// LS Electric XG5000 project: Test1108
// PLC NewPLC
// module base 0 slot 0: 입출력 모듈:XBC-DR32H (DC 24V 입력, 릴레이 출력 32점)

PROGRAM NewProgram (task: 스캔 프로그램)

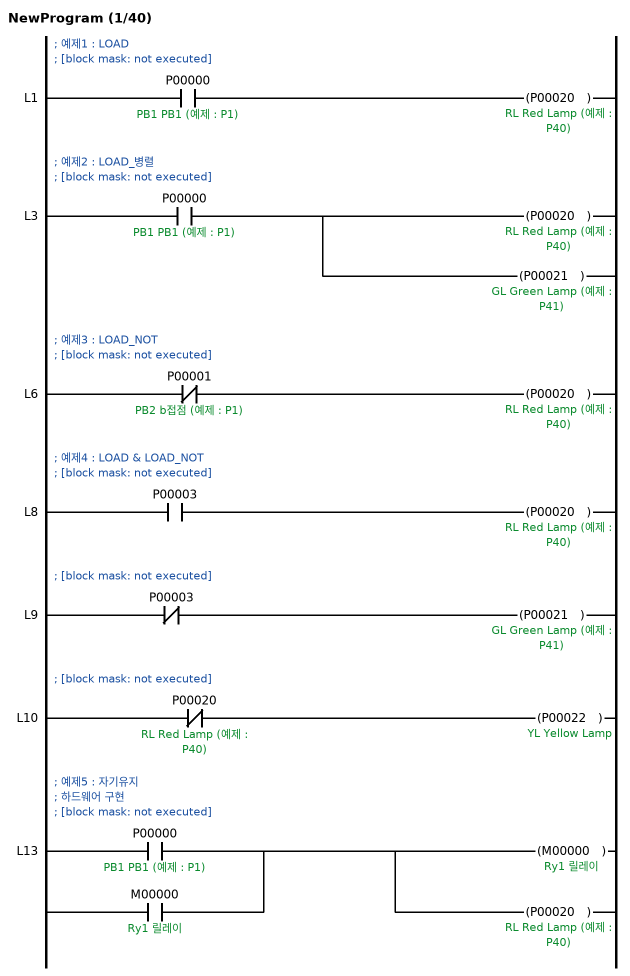
// 예제1 : LOAD
; L1 (block mask: not executed)
LOAD      P00000	// PB1 PB1 (예제 : P1)
OUT       P00020	// RL Red Lamp (예제 : P40)
// 예제2 : LOAD_병렬
; L3 (block mask: not executed)
LOAD      P00000	// PB1 PB1 (예제 : P1)
OUT       P00020	// RL Red Lamp (예제 : P40)
OUT       P00021	// GL Green Lamp (예제 : P41)
// 예제3 : LOAD_NOT 
; L6 (block mask: not executed)
LOAD NOT  P00001	// PB2 b접점 (예제 : P1)
OUT       P00020	// RL Red Lamp (예제 : P40)
// 예제4 : LOAD & LOAD_NOT
; L8 (block mask: not executed)
LOAD      P00003
OUT       P00020	// RL Red Lamp (예제 : P40)
; L9 (block mask: not executed)
LOAD NOT  P00003
OUT       P00021	// GL Green Lamp (예제 : P41)
; L10 (block mask: not executed)
LOAD NOT  P00020	// RL Red Lamp (예제 : P40)
OUT       P00022	// YL Yellow Lamp
// 예제5 : 자기유지
// 하드웨어 구현
; L13 (block mask: not executed)
LOAD      P00000	// PB1 PB1 (예제 : P1)
OR        M00000	// Ry1 릴레이
OUT       M00000	// Ry1 릴레이
OUT       P00020	// RL Red Lamp (예제 : P40)

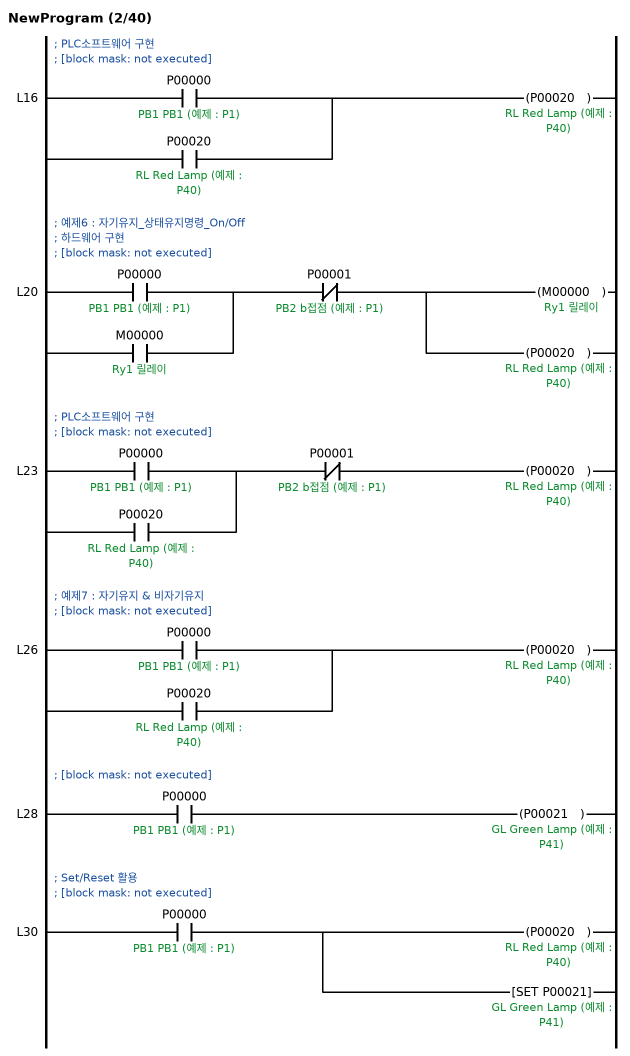
// PLC소프트웨어 구현
; L16 (block mask: not executed)
LOAD      P00000	// PB1 PB1 (예제 : P1)
OR        P00020	// RL Red Lamp (예제 : P40)
OUT       P00020	// RL Red Lamp (예제 : P40)
// 예제6 : 자기유지_상태유지명령_On/Off
// 하드웨어 구현
; L20 (block mask: not executed)
LOAD      P00000	// PB1 PB1 (예제 : P1)
OR        M00000	// Ry1 릴레이
AND NOT   P00001	// PB2 b접점 (예제 : P1)
OUT       M00000	// Ry1 릴레이
OUT       P00020	// RL Red Lamp (예제 : P40)
// PLC소프트웨어 구현
; L23 (block mask: not executed)
LOAD      P00000	// PB1 PB1 (예제 : P1)
OR        P00020	// RL Red Lamp (예제 : P40)
AND NOT   P00001	// PB2 b접점 (예제 : P1)
OUT       P00020	// RL Red Lamp (예제 : P40)
// 예제7 : 자기유지 & 비자기유지
; L26 (block mask: not executed)
LOAD      P00000	// PB1 PB1 (예제 : P1)
OR        P00020	// RL Red Lamp (예제 : P40)
OUT       P00020	// RL Red Lamp (예제 : P40)
; L28 (block mask: not executed)
LOAD      P00000	// PB1 PB1 (예제 : P1)
OUT       P00021	// GL Green Lamp (예제 : P41)
// Set/Reset 활용
; L30 (block mask: not executed)
LOAD      P00000	// PB1 PB1 (예제 : P1)
OUT       P00020	// RL Red Lamp (예제 : P40)
SET       P00021	// GL Green Lamp (예제 : P41)

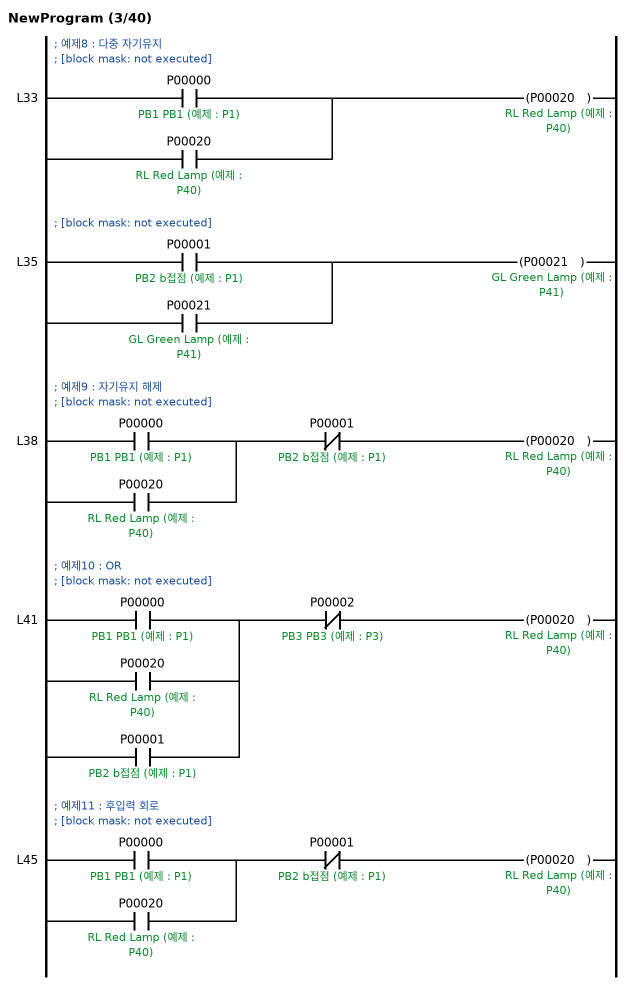
// 예제8 : 다중 자기유지
; L33 (block mask: not executed)
LOAD      P00000	// PB1 PB1 (예제 : P1)
OR        P00020	// RL Red Lamp (예제 : P40)
OUT       P00020	// RL Red Lamp (예제 : P40)
; L35 (block mask: not executed)
LOAD      P00001	// PB2 b접점 (예제 : P1)
OR        P00021	// GL Green Lamp (예제 : P41)
OUT       P00021	// GL Green Lamp (예제 : P41)
// 예제9 : 자기유지 해제
; L38 (block mask: not executed)
LOAD      P00000	// PB1 PB1 (예제 : P1)
OR        P00020	// RL Red Lamp (예제 : P40)
AND NOT   P00001	// PB2 b접점 (예제 : P1)
OUT       P00020	// RL Red Lamp (예제 : P40)
// 예제10 : OR
; L41 (block mask: not executed)
LOAD      P00000	// PB1 PB1 (예제 : P1)
OR        P00020	// RL Red Lamp (예제 : P40)
OR        P00001	// PB2 b접점 (예제 : P1)
AND NOT   P00002	// PB3 PB3 (예제 : P3)
OUT       P00020	// RL Red Lamp (예제 : P40)
// 예제11 : 후입력 회로
; L45 (block mask: not executed)
LOAD      P00000	// PB1 PB1 (예제 : P1)
OR        P00020	// RL Red Lamp (예제 : P40)
AND NOT   P00001	// PB2 b접점 (예제 : P1)
OUT       P00020	// RL Red Lamp (예제 : P40)

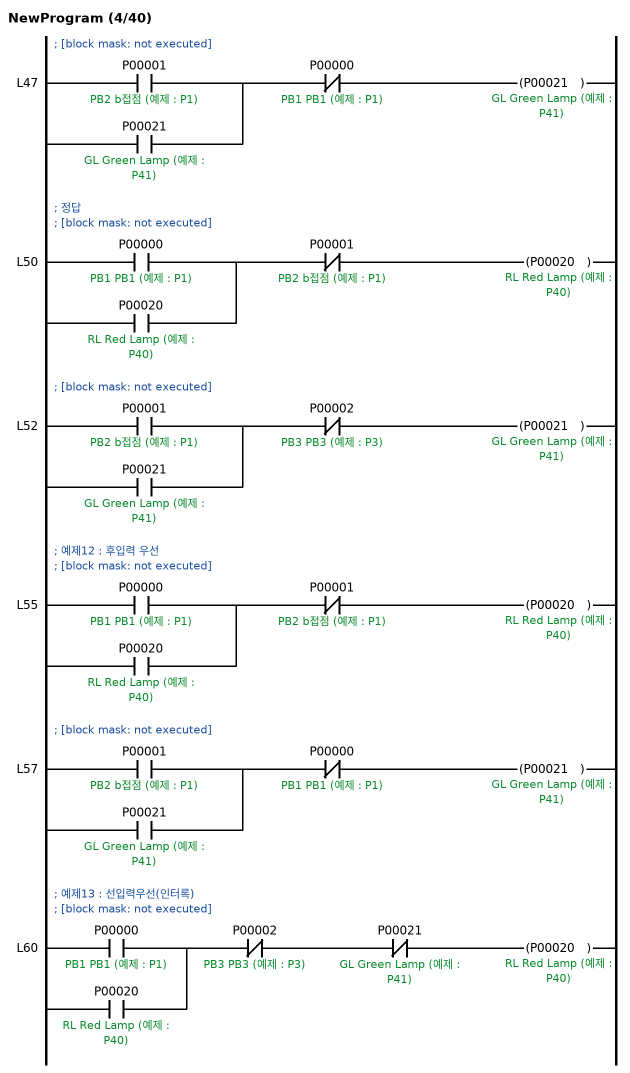
; L47 (block mask: not executed)
LOAD      P00001	// PB2 b접점 (예제 : P1)
OR        P00021	// GL Green Lamp (예제 : P41)
AND NOT   P00000	// PB1 PB1 (예제 : P1)
OUT       P00021	// GL Green Lamp (예제 : P41)
// 정답
; L50 (block mask: not executed)
LOAD      P00000	// PB1 PB1 (예제 : P1)
OR        P00020	// RL Red Lamp (예제 : P40)
AND NOT   P00001	// PB2 b접점 (예제 : P1)
OUT       P00020	// RL Red Lamp (예제 : P40)
; L52 (block mask: not executed)
LOAD      P00001	// PB2 b접점 (예제 : P1)
OR        P00021	// GL Green Lamp (예제 : P41)
AND NOT   P00002	// PB3 PB3 (예제 : P3)
OUT       P00021	// GL Green Lamp (예제 : P41)
// 예제12 : 후입력 우선
; L55 (block mask: not executed)
LOAD      P00000	// PB1 PB1 (예제 : P1)
OR        P00020	// RL Red Lamp (예제 : P40)
AND NOT   P00001	// PB2 b접점 (예제 : P1)
OUT       P00020	// RL Red Lamp (예제 : P40)
; L57 (block mask: not executed)
LOAD      P00001	// PB2 b접점 (예제 : P1)
OR        P00021	// GL Green Lamp (예제 : P41)
AND NOT   P00000	// PB1 PB1 (예제 : P1)
OUT       P00021	// GL Green Lamp (예제 : P41)
// 예제13 : 선입력우선(인터록)
; L60 (block mask: not executed)
LOAD      P00000	// PB1 PB1 (예제 : P1)
OR        P00020	// RL Red Lamp (예제 : P40)
AND NOT   P00002	// PB3 PB3 (예제 : P3)
AND NOT   P00021	// GL Green Lamp (예제 : P41)
OUT       P00020	// RL Red Lamp (예제 : P40)

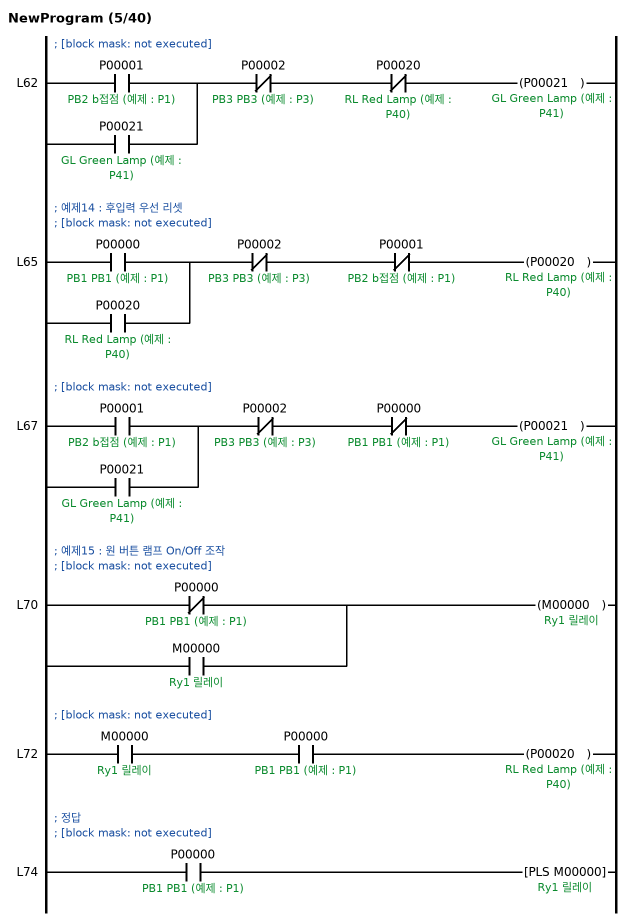
; L62 (block mask: not executed)
LOAD      P00001	// PB2 b접점 (예제 : P1)
OR        P00021	// GL Green Lamp (예제 : P41)
AND NOT   P00002	// PB3 PB3 (예제 : P3)
AND NOT   P00020	// RL Red Lamp (예제 : P40)
OUT       P00021	// GL Green Lamp (예제 : P41)
// 예제14 : 후입력 우선 리셋
; L65 (block mask: not executed)
LOAD      P00000	// PB1 PB1 (예제 : P1)
OR        P00020	// RL Red Lamp (예제 : P40)
AND NOT   P00002	// PB3 PB3 (예제 : P3)
AND NOT   P00001	// PB2 b접점 (예제 : P1)
OUT       P00020	// RL Red Lamp (예제 : P40)
; L67 (block mask: not executed)
LOAD      P00001	// PB2 b접점 (예제 : P1)
OR        P00021	// GL Green Lamp (예제 : P41)
AND NOT   P00002	// PB3 PB3 (예제 : P3)
AND NOT   P00000	// PB1 PB1 (예제 : P1)
OUT       P00021	// GL Green Lamp (예제 : P41)
// 예제15 : 원 버튼 램프 On/Off 조작
; L70 (block mask: not executed)
LOAD NOT  P00000	// PB1 PB1 (예제 : P1)
OR        M00000	// Ry1 릴레이
OUT       M00000	// Ry1 릴레이
; L72 (block mask: not executed)
LOAD      M00000	// Ry1 릴레이
AND       P00000	// PB1 PB1 (예제 : P1)
OUT       P00020	// RL Red Lamp (예제 : P40)
// 정답
; L74 (block mask: not executed)
LOAD      P00000	// PB1 PB1 (예제 : P1)
OUTP      M00000	// Ry1 릴레이

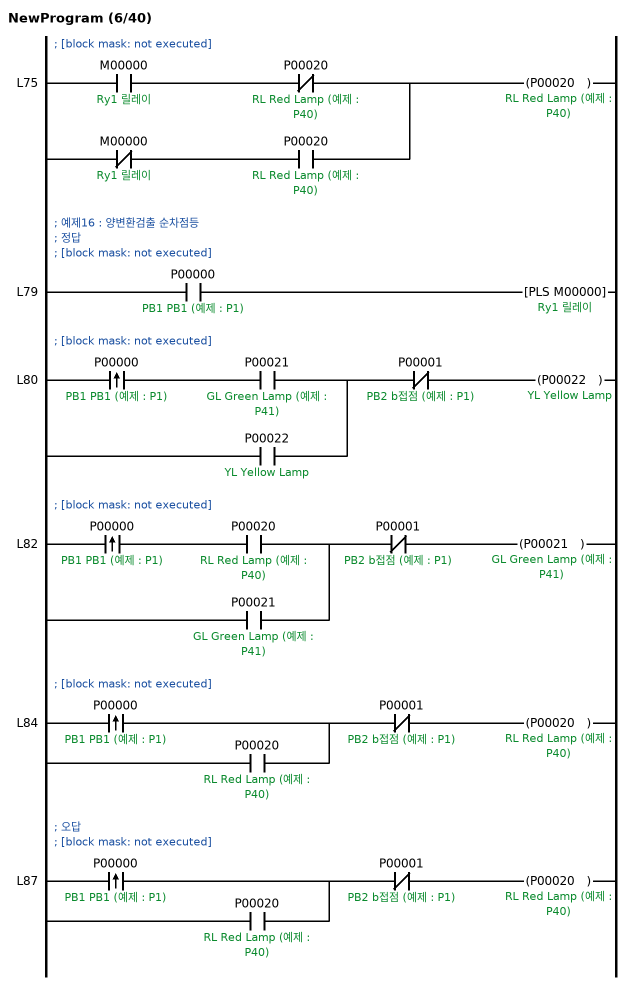
; L75 (block mask: not executed)
LOAD      M00000	// Ry1 릴레이
AND NOT   P00020	// RL Red Lamp (예제 : P40)
LOAD NOT  M00000	// Ry1 릴레이
AND       P00020	// RL Red Lamp (예제 : P40)
OR LOAD
OUT       P00020	// RL Red Lamp (예제 : P40)
// 예제16 : 양변환검출 순차점등
// 정답
; L79 (block mask: not executed)
LOAD      P00000	// PB1 PB1 (예제 : P1)
OUTP      M00000	// Ry1 릴레이
; L80 (block mask: not executed)
LOADP     P00000	// PB1 PB1 (예제 : P1)
AND       P00021	// GL Green Lamp (예제 : P41)
OR        P00022	// YL Yellow Lamp
AND NOT   P00001	// PB2 b접점 (예제 : P1)
OUT       P00022	// YL Yellow Lamp
; L82 (block mask: not executed)
LOADP     P00000	// PB1 PB1 (예제 : P1)
AND       P00020	// RL Red Lamp (예제 : P40)
OR        P00021	// GL Green Lamp (예제 : P41)
AND NOT   P00001	// PB2 b접점 (예제 : P1)
OUT       P00021	// GL Green Lamp (예제 : P41)
; L84 (block mask: not executed)
LOADP     P00000	// PB1 PB1 (예제 : P1)
OR        P00020	// RL Red Lamp (예제 : P40)
AND NOT   P00001	// PB2 b접점 (예제 : P1)
OUT       P00020	// RL Red Lamp (예제 : P40)
// 오답
; L87 (block mask: not executed)
LOADP     P00000	// PB1 PB1 (예제 : P1)
OR        P00020	// RL Red Lamp (예제 : P40)
AND NOT   P00001	// PB2 b접점 (예제 : P1)
OUT       P00020	// RL Red Lamp (예제 : P40)

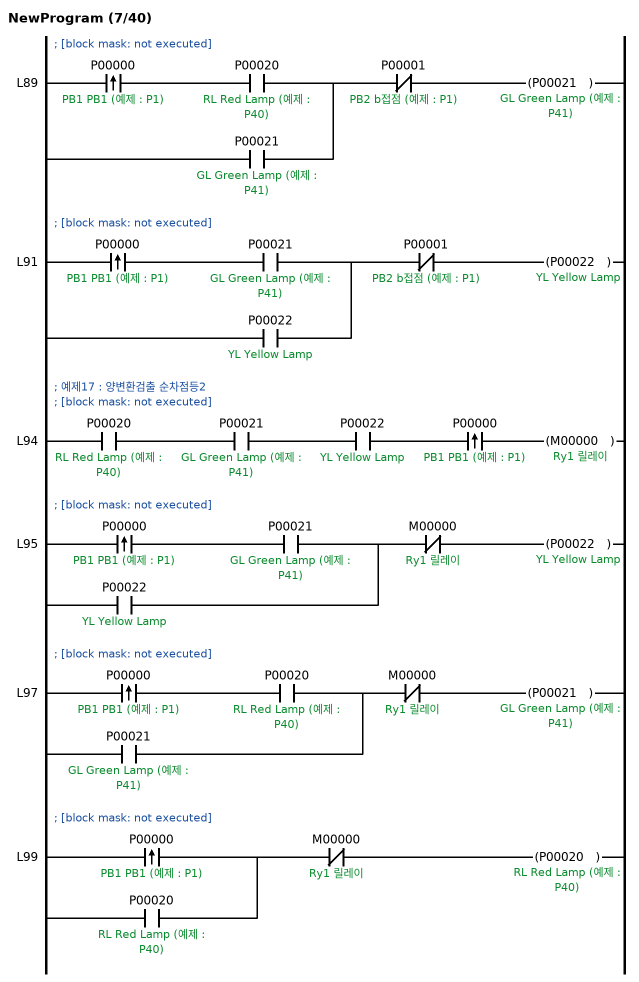
; L89 (block mask: not executed)
LOADP     P00000	// PB1 PB1 (예제 : P1)
AND       P00020	// RL Red Lamp (예제 : P40)
OR        P00021	// GL Green Lamp (예제 : P41)
AND NOT   P00001	// PB2 b접점 (예제 : P1)
OUT       P00021	// GL Green Lamp (예제 : P41)
; L91 (block mask: not executed)
LOADP     P00000	// PB1 PB1 (예제 : P1)
AND       P00021	// GL Green Lamp (예제 : P41)
OR        P00022	// YL Yellow Lamp
AND NOT   P00001	// PB2 b접점 (예제 : P1)
OUT       P00022	// YL Yellow Lamp
// 예제17 : 양변환검출 순차점등2
; L94 (block mask: not executed)
LOAD      P00020	// RL Red Lamp (예제 : P40)
AND       P00021	// GL Green Lamp (예제 : P41)
AND       P00022	// YL Yellow Lamp
ANDP      P00000	// PB1 PB1 (예제 : P1)
OUT       M00000	// Ry1 릴레이
; L95 (block mask: not executed)
LOADP     P00000	// PB1 PB1 (예제 : P1)
AND       P00021	// GL Green Lamp (예제 : P41)
OR        P00022	// YL Yellow Lamp
AND NOT   M00000	// Ry1 릴레이
OUT       P00022	// YL Yellow Lamp
; L97 (block mask: not executed)
LOADP     P00000	// PB1 PB1 (예제 : P1)
AND       P00020	// RL Red Lamp (예제 : P40)
OR        P00021	// GL Green Lamp (예제 : P41)
AND NOT   M00000	// Ry1 릴레이
OUT       P00021	// GL Green Lamp (예제 : P41)
; L99 (block mask: not executed)
LOADP     P00000	// PB1 PB1 (예제 : P1)
OR        P00020	// RL Red Lamp (예제 : P40)
AND NOT   M00000	// Ry1 릴레이
OUT       P00020	// RL Red Lamp (예제 : P40)

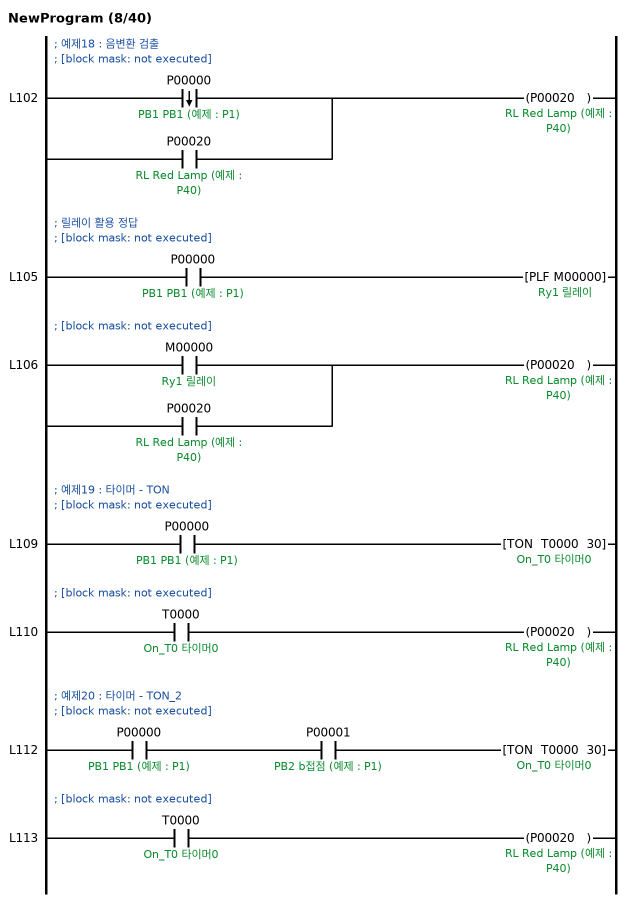
// 예제18 : 음변환 검출
; L102 (block mask: not executed)
LOADN     P00000	// PB1 PB1 (예제 : P1)
OR        P00020	// RL Red Lamp (예제 : P40)
OUT       P00020	// RL Red Lamp (예제 : P40)
// 릴레이 활용 정답
; L105 (block mask: not executed)
LOAD      P00000	// PB1 PB1 (예제 : P1)
OUTN      M00000	// Ry1 릴레이
; L106 (block mask: not executed)
LOAD      M00000	// Ry1 릴레이
OR        P00020	// RL Red Lamp (예제 : P40)
OUT       P00020	// RL Red Lamp (예제 : P40)
// 예제19 : 타이머 - TON
; L109 (block mask: not executed)
LOAD      P00000	// PB1 PB1 (예제 : P1)
TON       T0000 30	// On_T0 타이머0
; L110 (block mask: not executed)
LOAD      T0000	// On_T0 타이머0
OUT       P00020	// RL Red Lamp (예제 : P40)
// 예제20 : 타이머 - TON_2
; L112 (block mask: not executed)
LOAD      P00000	// PB1 PB1 (예제 : P1)
AND       P00001	// PB2 b접점 (예제 : P1)
TON       T0000 30	// On_T0 타이머0
; L113 (block mask: not executed)
LOAD      T0000	// On_T0 타이머0
OUT       P00020	// RL Red Lamp (예제 : P40)

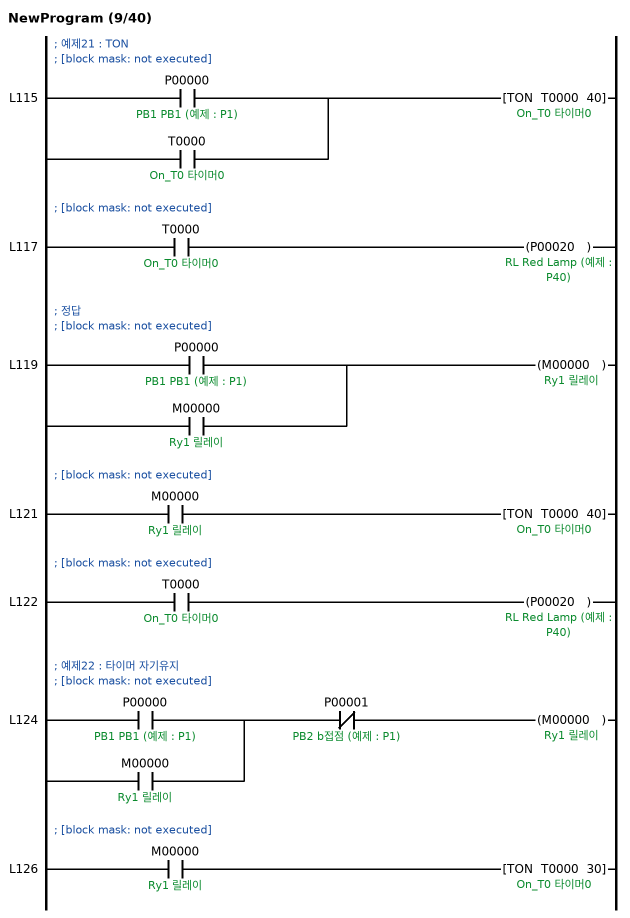
// 예제21 : TON
; L115 (block mask: not executed)
LOAD      P00000	// PB1 PB1 (예제 : P1)
OR        T0000	// On_T0 타이머0
TON       T0000 40	// On_T0 타이머0
; L117 (block mask: not executed)
LOAD      T0000	// On_T0 타이머0
OUT       P00020	// RL Red Lamp (예제 : P40)
// 정답
; L119 (block mask: not executed)
LOAD      P00000	// PB1 PB1 (예제 : P1)
OR        M00000	// Ry1 릴레이
OUT       M00000	// Ry1 릴레이
; L121 (block mask: not executed)
LOAD      M00000	// Ry1 릴레이
TON       T0000 40	// On_T0 타이머0
; L122 (block mask: not executed)
LOAD      T0000	// On_T0 타이머0
OUT       P00020	// RL Red Lamp (예제 : P40)
// 예제22 : 타이머 자기유지
; L124 (block mask: not executed)
LOAD      P00000	// PB1 PB1 (예제 : P1)
OR        M00000	// Ry1 릴레이
AND NOT   P00001	// PB2 b접점 (예제 : P1)
OUT       M00000	// Ry1 릴레이
; L126 (block mask: not executed)
LOAD      M00000	// Ry1 릴레이
TON       T0000 30	// On_T0 타이머0

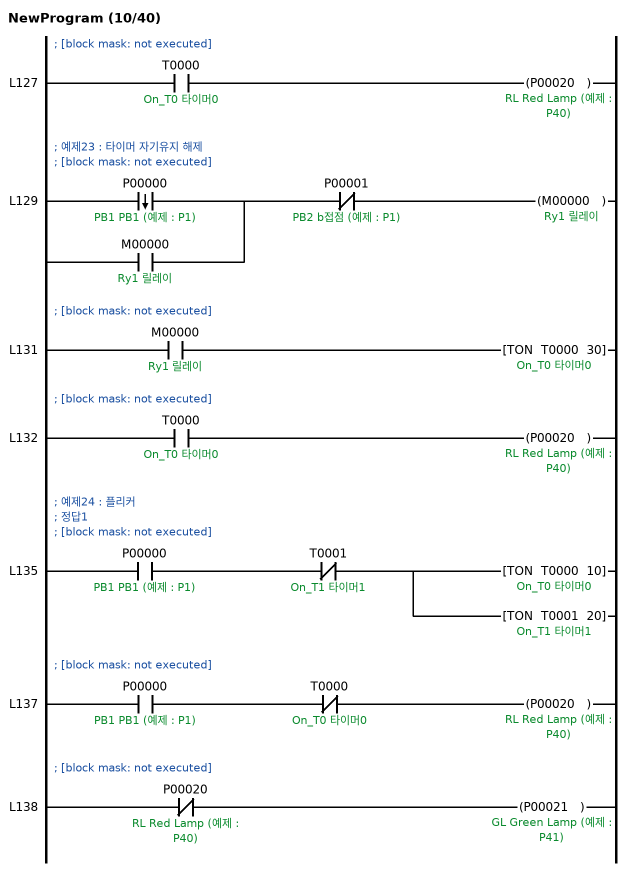
; L127 (block mask: not executed)
LOAD      T0000	// On_T0 타이머0
OUT       P00020	// RL Red Lamp (예제 : P40)
// 예제23 : 타이머 자기유지 해제
; L129 (block mask: not executed)
LOADN     P00000	// PB1 PB1 (예제 : P1)
OR        M00000	// Ry1 릴레이
AND NOT   P00001	// PB2 b접점 (예제 : P1)
OUT       M00000	// Ry1 릴레이
; L131 (block mask: not executed)
LOAD      M00000	// Ry1 릴레이
TON       T0000 30	// On_T0 타이머0
; L132 (block mask: not executed)
LOAD      T0000	// On_T0 타이머0
OUT       P00020	// RL Red Lamp (예제 : P40)
// 예제24 : 플리커
// 정답1
; L135 (block mask: not executed)
LOAD      P00000	// PB1 PB1 (예제 : P1)
AND NOT   T0001	// On_T1 타이머1
TON       T0000 10	// On_T0 타이머0
TON       T0001 20	// On_T1 타이머1
; L137 (block mask: not executed)
LOAD      P00000	// PB1 PB1 (예제 : P1)
AND NOT   T0000	// On_T0 타이머0
OUT       P00020	// RL Red Lamp (예제 : P40)
; L138 (block mask: not executed)
LOAD NOT  P00020	// RL Red Lamp (예제 : P40)
OUT       P00021	// GL Green Lamp (예제 : P41)

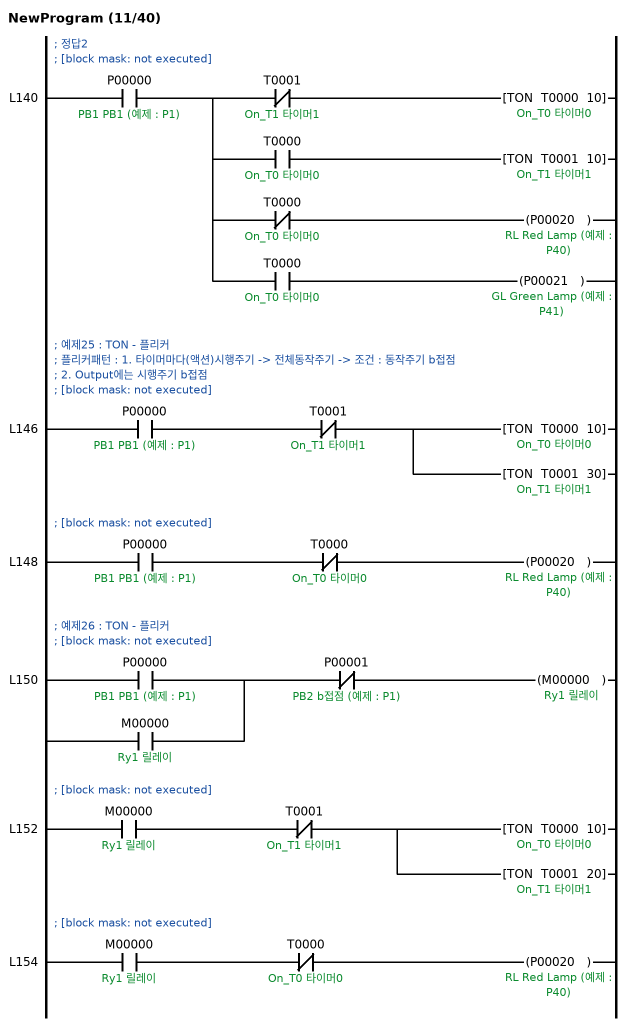
// 정답2
; L140 (block mask: not executed)
LOAD      P00000	// PB1 PB1 (예제 : P1)
MPUSH
AND NOT   T0001	// On_T1 타이머1
TON       T0000 10	// On_T0 타이머0
MLOAD
AND       T0000	// On_T0 타이머0
TON       T0001 10	// On_T1 타이머1
MLOAD
AND NOT   T0000	// On_T0 타이머0
OUT       P00020	// RL Red Lamp (예제 : P40)
MPOP
AND       T0000	// On_T0 타이머0
OUT       P00021	// GL Green Lamp (예제 : P41)
// 예제25 : TON - 플리커
// 플리커패턴 : 1. 타이머마다(액션)시행주기 -> 전체동작주기 -> 조건 : 동작주기 b접점 
//              2. Output에는 시행주기 b접점
; L146 (block mask: not executed)
LOAD      P00000	// PB1 PB1 (예제 : P1)
AND NOT   T0001	// On_T1 타이머1
TON       T0000 10	// On_T0 타이머0
TON       T0001 30	// On_T1 타이머1
; L148 (block mask: not executed)
LOAD      P00000	// PB1 PB1 (예제 : P1)
AND NOT   T0000	// On_T0 타이머0
OUT       P00020	// RL Red Lamp (예제 : P40)
// 예제26 : TON - 플리커
; L150 (block mask: not executed)
LOAD      P00000	// PB1 PB1 (예제 : P1)
OR        M00000	// Ry1 릴레이
AND NOT   P00001	// PB2 b접점 (예제 : P1)
OUT       M00000	// Ry1 릴레이
; L152 (block mask: not executed)
LOAD      M00000	// Ry1 릴레이
AND NOT   T0001	// On_T1 타이머1
TON       T0000 10	// On_T0 타이머0
TON       T0001 20	// On_T1 타이머1
; L154 (block mask: not executed)
LOAD      M00000	// Ry1 릴레이
AND NOT   T0000	// On_T0 타이머0
OUT       P00020	// RL Red Lamp (예제 : P40)

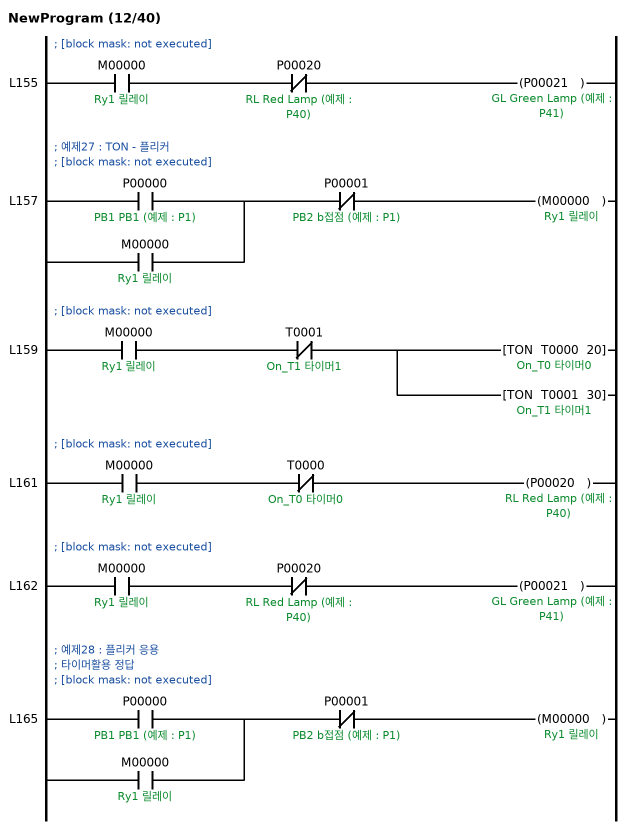
; L155 (block mask: not executed)
LOAD      M00000	// Ry1 릴레이
AND NOT   P00020	// RL Red Lamp (예제 : P40)
OUT       P00021	// GL Green Lamp (예제 : P41)
// 예제27 : TON - 플리커
; L157 (block mask: not executed)
LOAD      P00000	// PB1 PB1 (예제 : P1)
OR        M00000	// Ry1 릴레이
AND NOT   P00001	// PB2 b접점 (예제 : P1)
OUT       M00000	// Ry1 릴레이
; L159 (block mask: not executed)
LOAD      M00000	// Ry1 릴레이
AND NOT   T0001	// On_T1 타이머1
TON       T0000 20	// On_T0 타이머0
TON       T0001 30	// On_T1 타이머1
; L161 (block mask: not executed)
LOAD      M00000	// Ry1 릴레이
AND NOT   T0000	// On_T0 타이머0
OUT       P00020	// RL Red Lamp (예제 : P40)
; L162 (block mask: not executed)
LOAD      M00000	// Ry1 릴레이
AND NOT   P00020	// RL Red Lamp (예제 : P40)
OUT       P00021	// GL Green Lamp (예제 : P41)
// 예제28 : 플리커 응용
// 타이머활용 정답
; L165 (block mask: not executed)
LOAD      P00000	// PB1 PB1 (예제 : P1)
OR        M00000	// Ry1 릴레이
AND NOT   P00001	// PB2 b접점 (예제 : P1)
OUT       M00000	// Ry1 릴레이

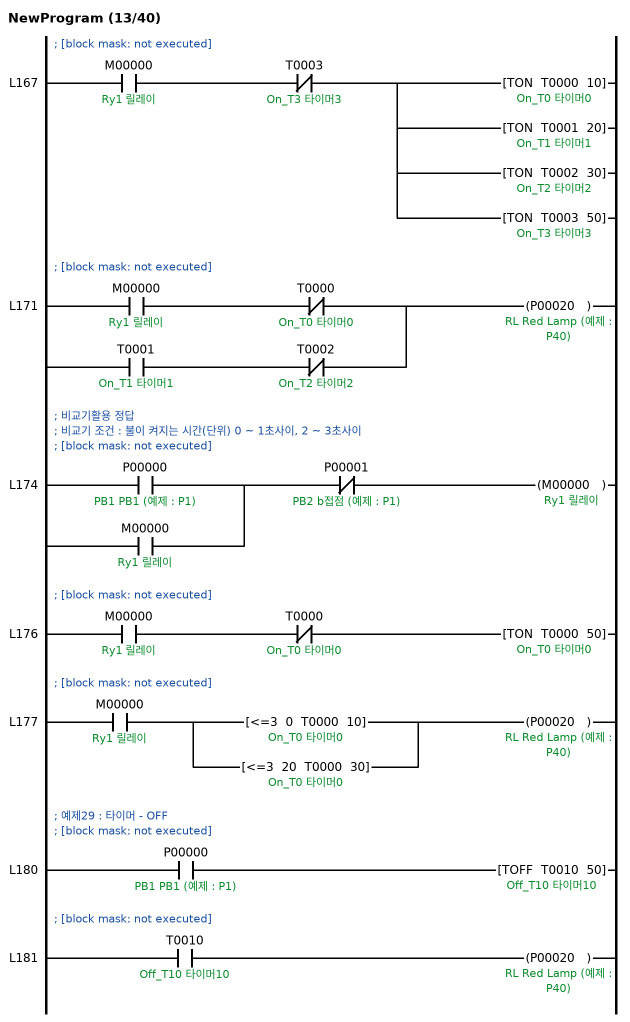
; L167 (block mask: not executed)
LOAD      M00000	// Ry1 릴레이
AND NOT   T0003	// On_T3 타이머3
TON       T0000 10	// On_T0 타이머0
TON       T0001 20	// On_T1 타이머1
TON       T0002 30	// On_T2 타이머2
TON       T0003 50	// On_T3 타이머3
; L171 (block mask: not executed)
LOAD      M00000	// Ry1 릴레이
AND NOT   T0000	// On_T0 타이머0
LOAD      T0001	// On_T1 타이머1
AND NOT   T0002	// On_T2 타이머2
OR LOAD
OUT       P00020	// RL Red Lamp (예제 : P40)
// 비교기활용 정답
//  비교기 조건 : 불이 켜지는 시간(단위) 0 ~ 1초사이, 2 ~ 3초사이
; L174 (block mask: not executed)
LOAD      P00000	// PB1 PB1 (예제 : P1)
OR        M00000	// Ry1 릴레이
AND NOT   P00001	// PB2 b접점 (예제 : P1)
OUT       M00000	// Ry1 릴레이
; L176 (block mask: not executed)
LOAD      M00000	// Ry1 릴레이
AND NOT   T0000	// On_T0 타이머0
TON       T0000 50	// On_T0 타이머0
; L177 (block mask: not executed)
LOAD      M00000	// Ry1 릴레이
LOAD<=3   0 T0000 10	// On_T0 타이머0
OR<=3     20 T0000 30	// On_T0 타이머0
AND LOAD
OUT       P00020	// RL Red Lamp (예제 : P40)
// 예제29 : 타이머 - OFF
; L180 (block mask: not executed)
LOAD      P00000	// PB1 PB1 (예제 : P1)
TOFF      T0010 50	// Off_T10 타이머10
; L181 (block mask: not executed)
LOAD      T0010	// Off_T10 타이머10
OUT       P00020	// RL Red Lamp (예제 : P40)

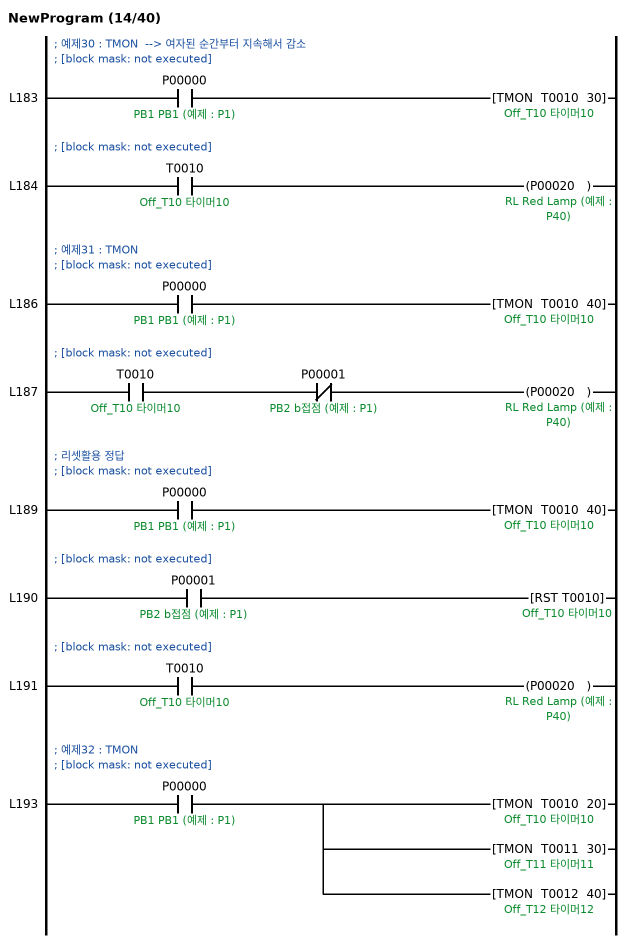
// 예제30 : TMON  --> 여자된 순간부터 지속해서 감소
; L183 (block mask: not executed)
LOAD      P00000	// PB1 PB1 (예제 : P1)
TMON      T0010 30	// Off_T10 타이머10
; L184 (block mask: not executed)
LOAD      T0010	// Off_T10 타이머10
OUT       P00020	// RL Red Lamp (예제 : P40)
// 예제31 : TMON
; L186 (block mask: not executed)
LOAD      P00000	// PB1 PB1 (예제 : P1)
TMON      T0010 40	// Off_T10 타이머10
; L187 (block mask: not executed)
LOAD      T0010	// Off_T10 타이머10
AND NOT   P00001	// PB2 b접점 (예제 : P1)
OUT       P00020	// RL Red Lamp (예제 : P40)
// 리셋활용 정답
; L189 (block mask: not executed)
LOAD      P00000	// PB1 PB1 (예제 : P1)
TMON      T0010 40	// Off_T10 타이머10
; L190 (block mask: not executed)
LOAD      P00001	// PB2 b접점 (예제 : P1)
RST       T0010	// Off_T10 타이머10
; L191 (block mask: not executed)
LOAD      T0010	// Off_T10 타이머10
OUT       P00020	// RL Red Lamp (예제 : P40)
// 예제32 : TMON
; L193 (block mask: not executed)
LOAD      P00000	// PB1 PB1 (예제 : P1)
TMON      T0010 20	// Off_T10 타이머10
TMON      T0011 30	// Off_T11 타이머11
TMON      T0012 40	// Off_T12 타이머12

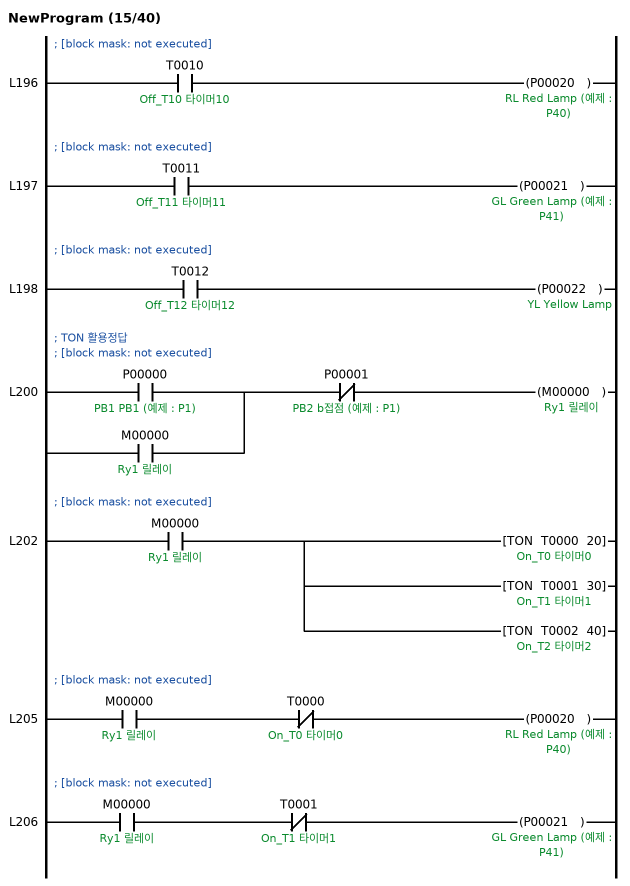
; L196 (block mask: not executed)
LOAD      T0010	// Off_T10 타이머10
OUT       P00020	// RL Red Lamp (예제 : P40)
; L197 (block mask: not executed)
LOAD      T0011	// Off_T11 타이머11
OUT       P00021	// GL Green Lamp (예제 : P41)
; L198 (block mask: not executed)
LOAD      T0012	// Off_T12 타이머12
OUT       P00022	// YL Yellow Lamp
// TON 활용정답
; L200 (block mask: not executed)
LOAD      P00000	// PB1 PB1 (예제 : P1)
OR        M00000	// Ry1 릴레이
AND NOT   P00001	// PB2 b접점 (예제 : P1)
OUT       M00000	// Ry1 릴레이
; L202 (block mask: not executed)
LOAD      M00000	// Ry1 릴레이
TON       T0000 20	// On_T0 타이머0
TON       T0001 30	// On_T1 타이머1
TON       T0002 40	// On_T2 타이머2
; L205 (block mask: not executed)
LOAD      M00000	// Ry1 릴레이
AND NOT   T0000	// On_T0 타이머0
OUT       P00020	// RL Red Lamp (예제 : P40)
; L206 (block mask: not executed)
LOAD      M00000	// Ry1 릴레이
AND NOT   T0001	// On_T1 타이머1
OUT       P00021	// GL Green Lamp (예제 : P41)

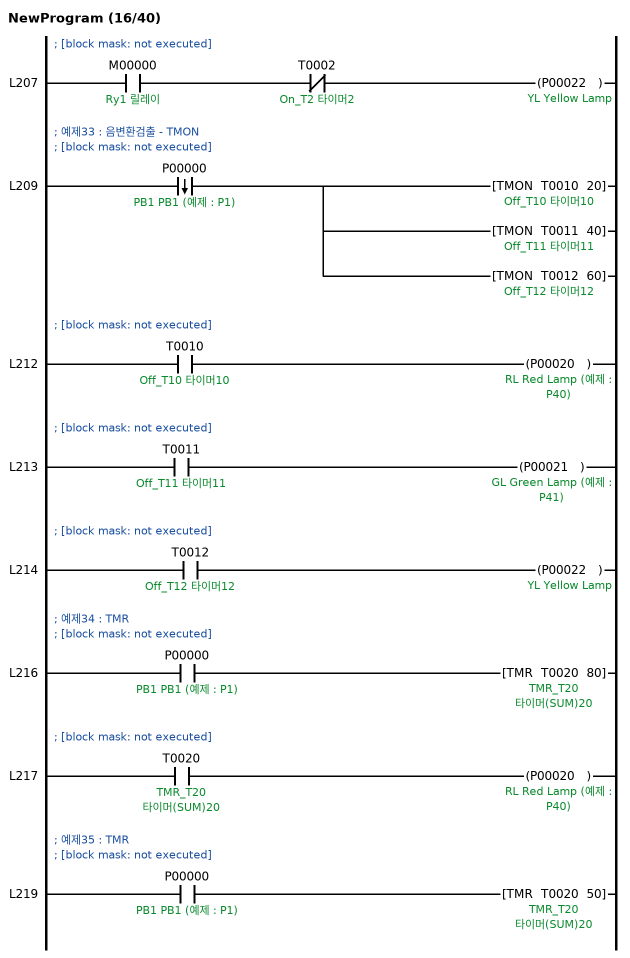
; L207 (block mask: not executed)
LOAD      M00000	// Ry1 릴레이
AND NOT   T0002	// On_T2 타이머2
OUT       P00022	// YL Yellow Lamp
// 예제33 : 음변환검출 - TMON
; L209 (block mask: not executed)
LOADN     P00000	// PB1 PB1 (예제 : P1)
TMON      T0010 20	// Off_T10 타이머10
TMON      T0011 40	// Off_T11 타이머11
TMON      T0012 60	// Off_T12 타이머12
; L212 (block mask: not executed)
LOAD      T0010	// Off_T10 타이머10
OUT       P00020	// RL Red Lamp (예제 : P40)
; L213 (block mask: not executed)
LOAD      T0011	// Off_T11 타이머11
OUT       P00021	// GL Green Lamp (예제 : P41)
; L214 (block mask: not executed)
LOAD      T0012	// Off_T12 타이머12
OUT       P00022	// YL Yellow Lamp
// 예제34 : TMR
; L216 (block mask: not executed)
LOAD      P00000	// PB1 PB1 (예제 : P1)
TMR       T0020 80	// TMR_T20 타이머(SUM)20
; L217 (block mask: not executed)
LOAD      T0020	// TMR_T20 타이머(SUM)20
OUT       P00020	// RL Red Lamp (예제 : P40)
// 예제35 : TMR
; L219 (block mask: not executed)
LOAD      P00000	// PB1 PB1 (예제 : P1)
TMR       T0020 50	// TMR_T20 타이머(SUM)20

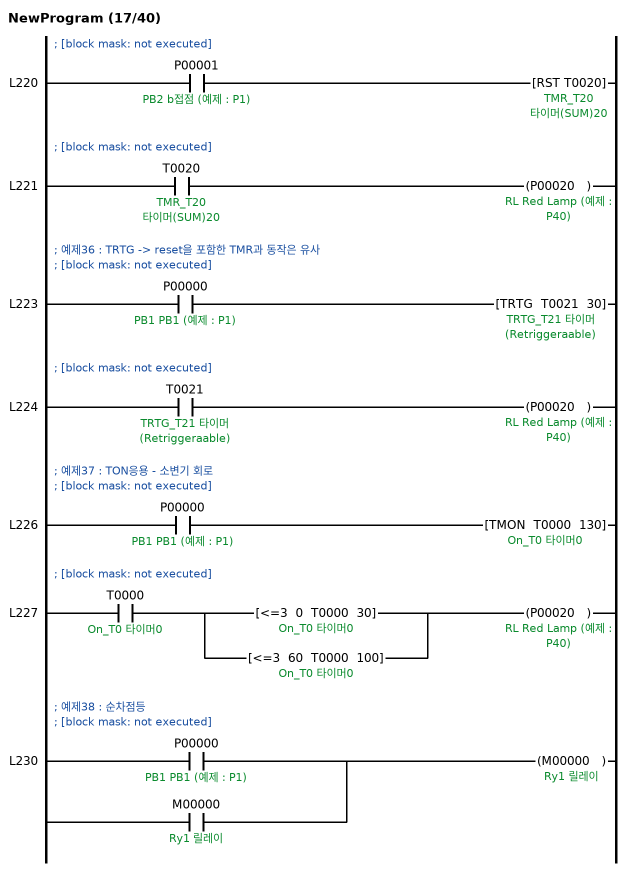
; L220 (block mask: not executed)
LOAD      P00001	// PB2 b접점 (예제 : P1)
RST       T0020	// TMR_T20 타이머(SUM)20
; L221 (block mask: not executed)
LOAD      T0020	// TMR_T20 타이머(SUM)20
OUT       P00020	// RL Red Lamp (예제 : P40)
// 예제36 : TRTG -> reset을 포함한 TMR과 동작은 유사
; L223 (block mask: not executed)
LOAD      P00000	// PB1 PB1 (예제 : P1)
TRTG      T0021 30	// TRTG_T21 타이머 (Retriggeraable)
; L224 (block mask: not executed)
LOAD      T0021	// TRTG_T21 타이머 (Retriggeraable)
OUT       P00020	// RL Red Lamp (예제 : P40)
// 예제37 : TON응용 - 소변기 회로
; L226 (block mask: not executed)
LOAD      P00000	// PB1 PB1 (예제 : P1)
TMON      T0000 130	// On_T0 타이머0
; L227 (block mask: not executed)
LOAD      T0000	// On_T0 타이머0
LOAD<=3   0 T0000 30	// On_T0 타이머0
OR<=3     60 T0000 100	// On_T0 타이머0
AND LOAD
OUT       P00020	// RL Red Lamp (예제 : P40)
// 예제38 : 순차점등
; L230 (block mask: not executed)
LOAD      P00000	// PB1 PB1 (예제 : P1)
OR        M00000	// Ry1 릴레이
OUT       M00000	// Ry1 릴레이

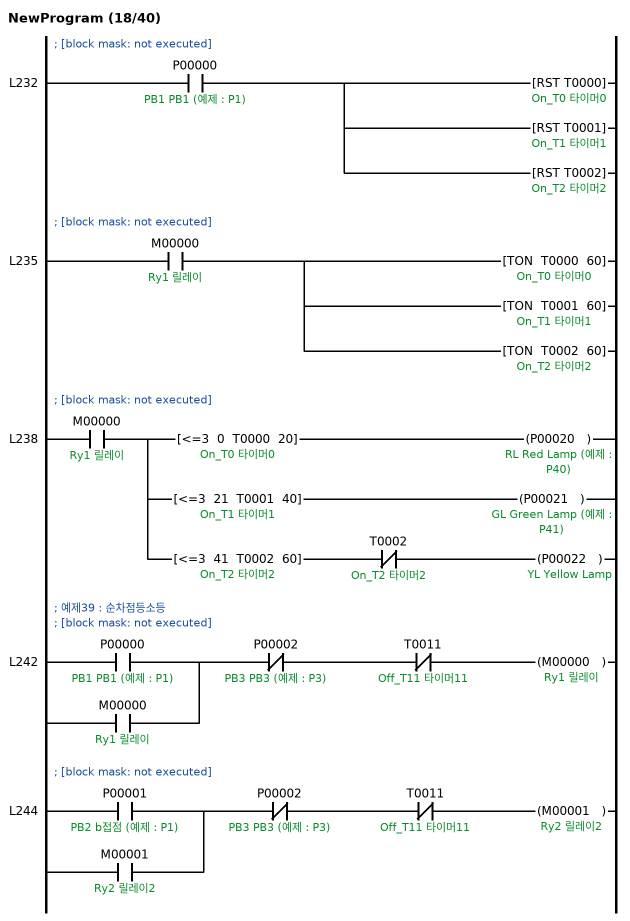
; L232 (block mask: not executed)
LOAD      P00000	// PB1 PB1 (예제 : P1)
RST       T0000	// On_T0 타이머0
RST       T0001	// On_T1 타이머1
RST       T0002	// On_T2 타이머2
; L235 (block mask: not executed)
LOAD      M00000	// Ry1 릴레이
TON       T0000 60	// On_T0 타이머0
TON       T0001 60	// On_T1 타이머1
TON       T0002 60	// On_T2 타이머2
; L238 (block mask: not executed)
LOAD      M00000	// Ry1 릴레이
MPUSH
AND<=3    0 T0000 20	// On_T0 타이머0
OUT       P00020	// RL Red Lamp (예제 : P40)
MLOAD
AND<=3    21 T0001 40	// On_T1 타이머1
OUT       P00021	// GL Green Lamp (예제 : P41)
MPOP
AND<=3    41 T0002 60	// On_T2 타이머2
AND NOT   T0002	// On_T2 타이머2
OUT       P00022	// YL Yellow Lamp
// 예제39 : 순차점등소등
; L242 (block mask: not executed)
LOAD      P00000	// PB1 PB1 (예제 : P1)
OR        M00000	// Ry1 릴레이
AND NOT   P00002	// PB3 PB3 (예제 : P3)
AND NOT   T0011	// Off_T11 타이머11
OUT       M00000	// Ry1 릴레이
; L244 (block mask: not executed)
LOAD      P00001	// PB2 b접점 (예제 : P1)
OR        M00001	// Ry2 릴레이2
AND NOT   P00002	// PB3 PB3 (예제 : P3)
AND NOT   T0011	// Off_T11 타이머11
OUT       M00001	// Ry2 릴레이2

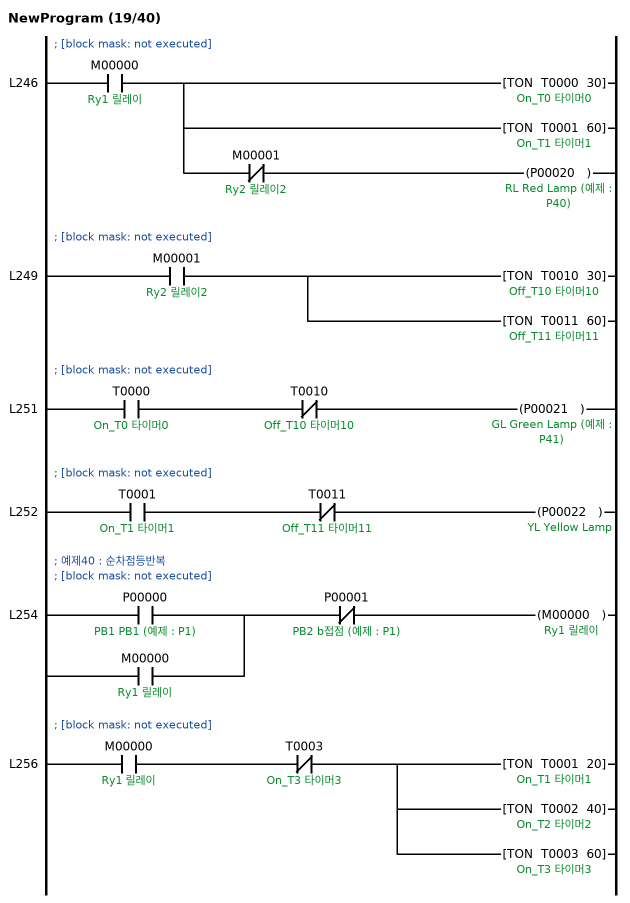
; L246 (block mask: not executed)
LOAD      M00000	// Ry1 릴레이
TON       T0000 30	// On_T0 타이머0
TON       T0001 60	// On_T1 타이머1
AND NOT   M00001	// Ry2 릴레이2
OUT       P00020	// RL Red Lamp (예제 : P40)
; L249 (block mask: not executed)
LOAD      M00001	// Ry2 릴레이2
TON       T0010 30	// Off_T10 타이머10
TON       T0011 60	// Off_T11 타이머11
; L251 (block mask: not executed)
LOAD      T0000	// On_T0 타이머0
AND NOT   T0010	// Off_T10 타이머10
OUT       P00021	// GL Green Lamp (예제 : P41)
; L252 (block mask: not executed)
LOAD      T0001	// On_T1 타이머1
AND NOT   T0011	// Off_T11 타이머11
OUT       P00022	// YL Yellow Lamp
// 예제40 : 순차점등반복
; L254 (block mask: not executed)
LOAD      P00000	// PB1 PB1 (예제 : P1)
OR        M00000	// Ry1 릴레이
AND NOT   P00001	// PB2 b접점 (예제 : P1)
OUT       M00000	// Ry1 릴레이
; L256 (block mask: not executed)
LOAD      M00000	// Ry1 릴레이
AND NOT   T0003	// On_T3 타이머3
TON       T0001 20	// On_T1 타이머1
TON       T0002 40	// On_T2 타이머2
TON       T0003 60	// On_T3 타이머3

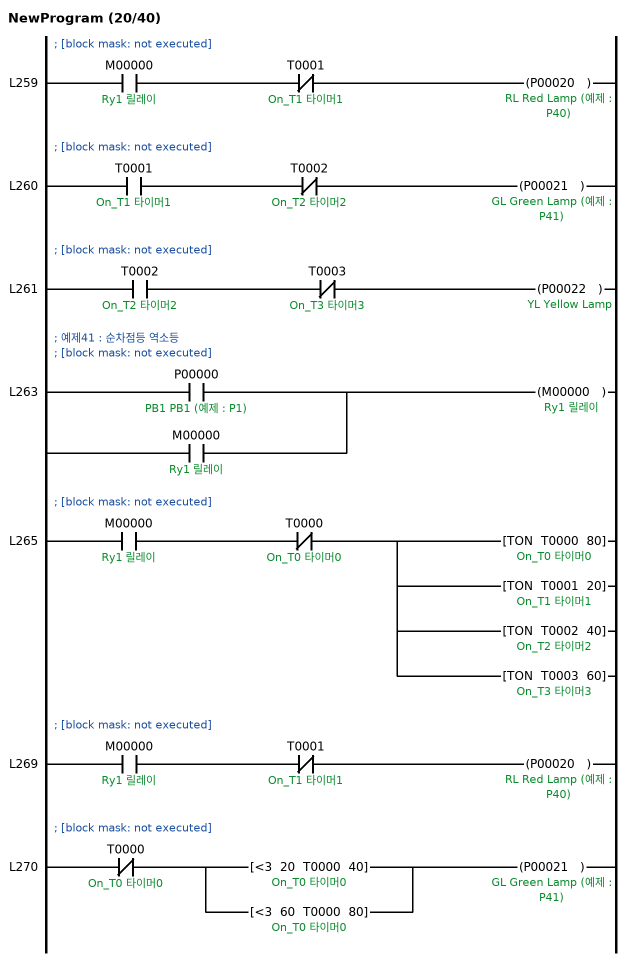
; L259 (block mask: not executed)
LOAD      M00000	// Ry1 릴레이
AND NOT   T0001	// On_T1 타이머1
OUT       P00020	// RL Red Lamp (예제 : P40)
; L260 (block mask: not executed)
LOAD      T0001	// On_T1 타이머1
AND NOT   T0002	// On_T2 타이머2
OUT       P00021	// GL Green Lamp (예제 : P41)
; L261 (block mask: not executed)
LOAD      T0002	// On_T2 타이머2
AND NOT   T0003	// On_T3 타이머3
OUT       P00022	// YL Yellow Lamp
// 예제41 : 순차점등 역소등
; L263 (block mask: not executed)
LOAD      P00000	// PB1 PB1 (예제 : P1)
OR        M00000	// Ry1 릴레이
OUT       M00000	// Ry1 릴레이
; L265 (block mask: not executed)
LOAD      M00000	// Ry1 릴레이
AND NOT   T0000	// On_T0 타이머0
TON       T0000 80	// On_T0 타이머0
TON       T0001 20	// On_T1 타이머1
TON       T0002 40	// On_T2 타이머2
TON       T0003 60	// On_T3 타이머3
; L269 (block mask: not executed)
LOAD      M00000	// Ry1 릴레이
AND NOT   T0001	// On_T1 타이머1
OUT       P00020	// RL Red Lamp (예제 : P40)
; L270 (block mask: not executed)
LOAD NOT  T0000	// On_T0 타이머0
LOAD<3    20 T0000 40	// On_T0 타이머0
OR<3      60 T0000 80	// On_T0 타이머0
AND LOAD
OUT       P00021	// GL Green Lamp (예제 : P41)

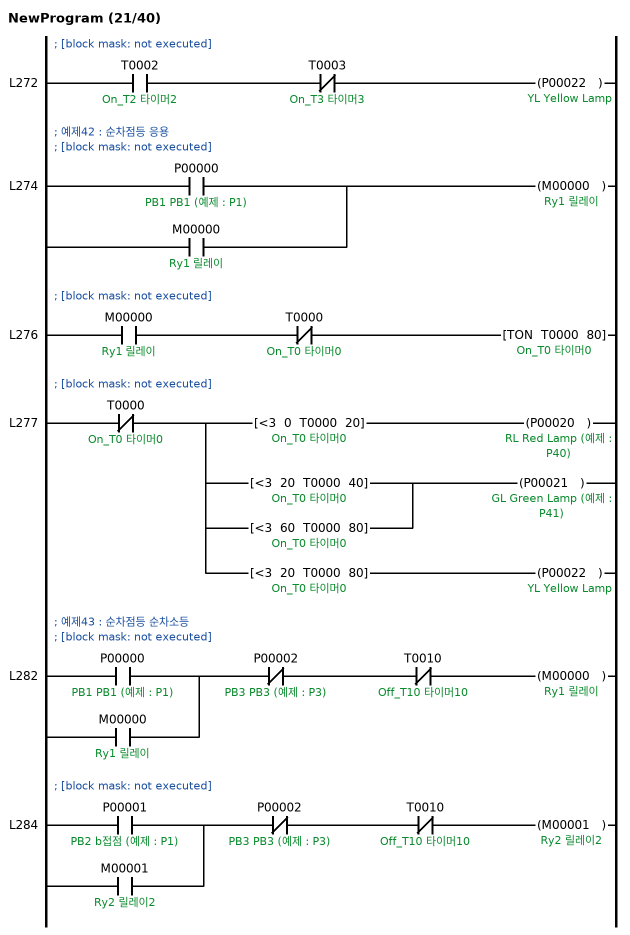
; L272 (block mask: not executed)
LOAD      T0002	// On_T2 타이머2
AND NOT   T0003	// On_T3 타이머3
OUT       P00022	// YL Yellow Lamp
// 예제42 : 순차점등 응용
; L274 (block mask: not executed)
LOAD      P00000	// PB1 PB1 (예제 : P1)
OR        M00000	// Ry1 릴레이
OUT       M00000	// Ry1 릴레이
; L276 (block mask: not executed)
LOAD      M00000	// Ry1 릴레이
AND NOT   T0000	// On_T0 타이머0
TON       T0000 80	// On_T0 타이머0
; L277 (block mask: not executed)
LOAD NOT  T0000	// On_T0 타이머0
MPUSH
AND<3     0 T0000 20	// On_T0 타이머0
OUT       P00020	// RL Red Lamp (예제 : P40)
MLOAD
LOAD<3    20 T0000 40	// On_T0 타이머0
OR<3      60 T0000 80	// On_T0 타이머0
AND LOAD
OUT       P00021	// GL Green Lamp (예제 : P41)
MPOP
AND<3     20 T0000 80	// On_T0 타이머0
OUT       P00022	// YL Yellow Lamp
// 예제43 : 순차점등 순차소등
; L282 (block mask: not executed)
LOAD      P00000	// PB1 PB1 (예제 : P1)
OR        M00000	// Ry1 릴레이
AND NOT   P00002	// PB3 PB3 (예제 : P3)
AND NOT   T0010	// Off_T10 타이머10
OUT       M00000	// Ry1 릴레이
; L284 (block mask: not executed)
LOAD      P00001	// PB2 b접점 (예제 : P1)
OR        M00001	// Ry2 릴레이2
AND NOT   P00002	// PB3 PB3 (예제 : P3)
AND NOT   T0010	// Off_T10 타이머10
OUT       M00001	// Ry2 릴레이2

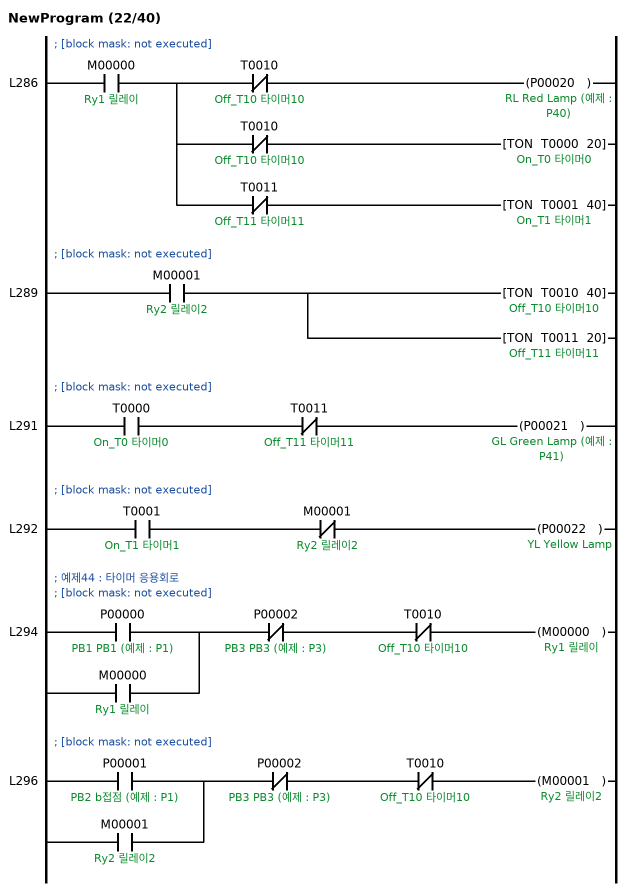
; L286 (block mask: not executed)
LOAD      M00000	// Ry1 릴레이
MPUSH
AND NOT   T0010	// Off_T10 타이머10
OUT       P00020	// RL Red Lamp (예제 : P40)
MLOAD
AND NOT   T0010	// Off_T10 타이머10
TON       T0000 20	// On_T0 타이머0
MPOP
AND NOT   T0011	// Off_T11 타이머11
TON       T0001 40	// On_T1 타이머1
; L289 (block mask: not executed)
LOAD      M00001	// Ry2 릴레이2
TON       T0010 40	// Off_T10 타이머10
TON       T0011 20	// Off_T11 타이머11
; L291 (block mask: not executed)
LOAD      T0000	// On_T0 타이머0
AND NOT   T0011	// Off_T11 타이머11
OUT       P00021	// GL Green Lamp (예제 : P41)
; L292 (block mask: not executed)
LOAD      T0001	// On_T1 타이머1
AND NOT   M00001	// Ry2 릴레이2
OUT       P00022	// YL Yellow Lamp
// 예제44 : 타이머 응용회로
; L294 (block mask: not executed)
LOAD      P00000	// PB1 PB1 (예제 : P1)
OR        M00000	// Ry1 릴레이
AND NOT   P00002	// PB3 PB3 (예제 : P3)
AND NOT   T0010	// Off_T10 타이머10
OUT       M00000	// Ry1 릴레이
; L296 (block mask: not executed)
LOAD      P00001	// PB2 b접점 (예제 : P1)
OR        M00001	// Ry2 릴레이2
AND NOT   P00002	// PB3 PB3 (예제 : P3)
AND NOT   T0010	// Off_T10 타이머10
OUT       M00001	// Ry2 릴레이2

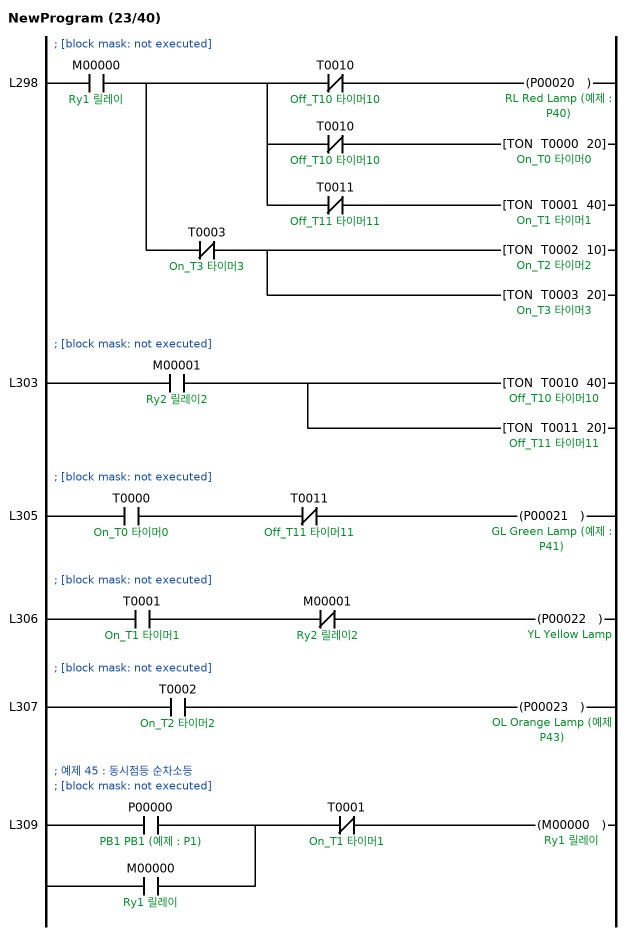
; L298 (block mask: not executed)
LOAD      M00000	// Ry1 릴레이
MPUSH
AND NOT   T0010	// Off_T10 타이머10
OUT       P00020	// RL Red Lamp (예제 : P40)
MLOAD
AND NOT   T0010	// Off_T10 타이머10
TON       T0000 20	// On_T0 타이머0
MLOAD
AND NOT   T0011	// Off_T11 타이머11
TON       T0001 40	// On_T1 타이머1
MPOP
AND NOT   T0003	// On_T3 타이머3
TON       T0002 10	// On_T2 타이머2
TON       T0003 20	// On_T3 타이머3
; L303 (block mask: not executed)
LOAD      M00001	// Ry2 릴레이2
TON       T0010 40	// Off_T10 타이머10
TON       T0011 20	// Off_T11 타이머11
; L305 (block mask: not executed)
LOAD      T0000	// On_T0 타이머0
AND NOT   T0011	// Off_T11 타이머11
OUT       P00021	// GL Green Lamp (예제 : P41)
; L306 (block mask: not executed)
LOAD      T0001	// On_T1 타이머1
AND NOT   M00001	// Ry2 릴레이2
OUT       P00022	// YL Yellow Lamp
; L307 (block mask: not executed)
LOAD      T0002	// On_T2 타이머2
OUT       P00023	// OL Orange Lamp (예제 P43)
// 예제 45 : 동시점등 순차소등
; L309 (block mask: not executed)
LOAD      P00000	// PB1 PB1 (예제 : P1)
OR        M00000	// Ry1 릴레이
AND NOT   T0001	// On_T1 타이머1
OUT       M00000	// Ry1 릴레이

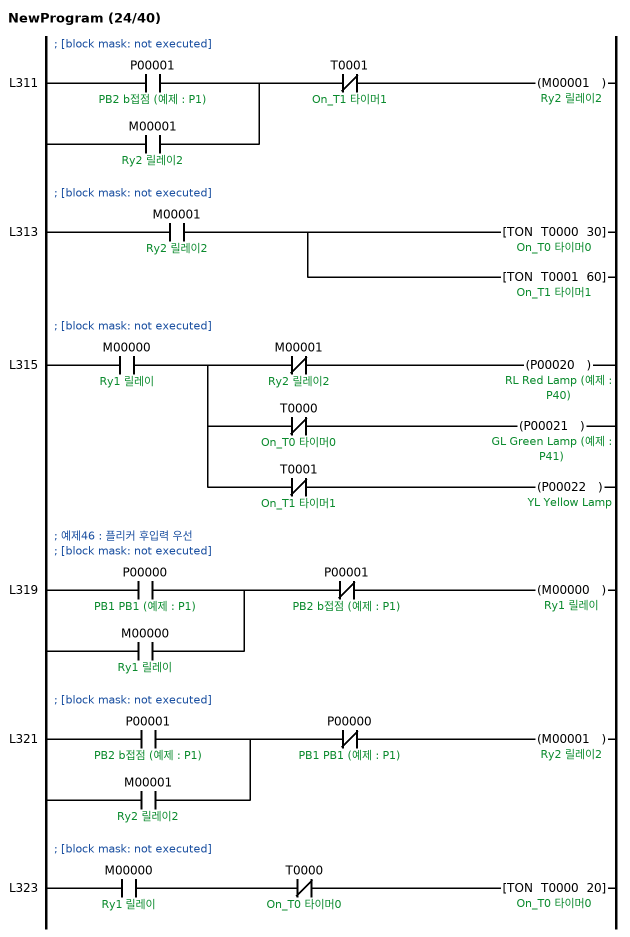
; L311 (block mask: not executed)
LOAD      P00001	// PB2 b접점 (예제 : P1)
OR        M00001	// Ry2 릴레이2
AND NOT   T0001	// On_T1 타이머1
OUT       M00001	// Ry2 릴레이2
; L313 (block mask: not executed)
LOAD      M00001	// Ry2 릴레이2
TON       T0000 30	// On_T0 타이머0
TON       T0001 60	// On_T1 타이머1
; L315 (block mask: not executed)
LOAD      M00000	// Ry1 릴레이
MPUSH
AND NOT   M00001	// Ry2 릴레이2
OUT       P00020	// RL Red Lamp (예제 : P40)
MLOAD
AND NOT   T0000	// On_T0 타이머0
OUT       P00021	// GL Green Lamp (예제 : P41)
MPOP
AND NOT   T0001	// On_T1 타이머1
OUT       P00022	// YL Yellow Lamp
// 예제46 : 플리커 후입력 우선
; L319 (block mask: not executed)
LOAD      P00000	// PB1 PB1 (예제 : P1)
OR        M00000	// Ry1 릴레이
AND NOT   P00001	// PB2 b접점 (예제 : P1)
OUT       M00000	// Ry1 릴레이
; L321 (block mask: not executed)
LOAD      P00001	// PB2 b접점 (예제 : P1)
OR        M00001	// Ry2 릴레이2
AND NOT   P00000	// PB1 PB1 (예제 : P1)
OUT       M00001	// Ry2 릴레이2
; L323 (block mask: not executed)
LOAD      M00000	// Ry1 릴레이
AND NOT   T0000	// On_T0 타이머0
TON       T0000 20	// On_T0 타이머0

